(* PLC project Untitled1, Beckhoff Automation GmbH TF6420 Database Server Query Analyser 1.0.0.0 *)
(* stored: creationDateTime 2020-05-15T10:13:58, modificationDateTime 2020-05-15T10:13:58 *)

TYPE 01_PCB_Ref : STRUCT
  Number : INT;
  Resistance : LREAL;
  Inductance : LREAL;
  Capacitance : LREAL;
END_STRUCT;
END_TYPE
